FUNCTION_BLOCK FB_MotorControl
VAR_INPUT
	Run 			: BOOL; // Order to start running
	Ready			: BOOL; // Safety ok, system ok, doors ok
	Fast 			: BOOL;
	Faster			: BOOL;
	VFD_Running		: BOOL;
	VFD_Ready		: BOOL;
END_VAR
VAR_OUTPUT
	Q : BOOL;
	RUN_Order_VFD 	: BOOL;
	Fast_VFD		: BOOL;
	Faster_VFD		: BOOL;
	iRounds 	: INT;
	iRoundsMinute : INT;
	Gato 		: BOOL;
	Perro 		: BOOL;
	GatoCount 	: INT;
	PerroCount 	: INT;
	iStatus		: INT;
	iFault		: INT;
END_VAR
VAR
	
	Run_TRIG: R_TRIG;
	nMotorState: (NOT_READY, ALL_READY, RUNNING, STOP, ERROR);
	SwitchLeft_TRIG: R_TRIG;
	SwitchRight_TRIG: R_TRIG;
	Stopping_TON: TON;
END_VAR

// Rough outline:
// INPUT 24V: DIB 4 5 6 eli paikat 14 15 16
// 4 käy/seis, 5 vakionopeus 1, 6 vakionopeus 2
// Taajarilta viestiä että joko on käynnissä tai valmis, ei tiedä vielä

// OUTPUT: 20, 24 25 26
// 20 = DO1, VALMIS-signaali
// 24-26 = rele, 25 vaihtaa paikkaa

// Kaukosäätimellä napilla käynnistyy ja pysähtyy (valo syttyy tai sammuu)
// Kytkimellä nopeus 1 tai 2 (vilkuttaa myös nopeammin tai hitaammin)

// Yksi anturi olisi pyörässä kiinni laskemassa kierroksia
// Valoanturi seuraamassa kun kissa tai koira menee ohi

// Valmius ja moottori käy/ei käy keskustelu taajarin kanssa joko digitaalilähdön kautta (valmius ehkä?) ja relelähdön kautta (miten toimikaan? Pitiköhän syöttää virtaa keskelle)
//Inputit vois Triguina yhä käsitellä, vaikka Buttonboxistakin tulee triguja. Mikäli jostain muusta lähteestä tulee käskyjä niin onpahan triguja yhä

//==================
// 7.10.22
// Moottori pyörii, käskyjä liikkuu. nyt erikoiskäyttö -profiili taajarissa, mutta EEPROM vika unohtaa kaikki asetukset.
// IN 1,2 on käy/suunta nyt, ei jaksa vaihtaa paremmaksi. 3 on Fast, mutta IN 4 ei ole taajarissa kytketty (sitten olisi Faster)
// OUT (taajarista) ei nopeasti katsoen rekisteröidy PLC:ssä. Relelähtö varmaan vääri kytketty


A_ButtonHandling();

CASE nMotorState OF
	NOT_READY:	
		Q := FALSE;
		IF Ready THEN
		nMotorState := 1;
		END_IF

	ALL_READY:
		IF NOT Ready THEN
			nMotorState := 0;
		END_IF 

		IF Run_TRIG.Q THEN
			Q := TRUE;
			nMotorState := 2;		
		END_IF
		
	RUNNING:
		IF NOT Ready THEN
			nMotorState := 0;
		END_IF 
		
		IF Run_TRIG.Q THEN
			Q := FALSE;
			nMotorState := 3;
		END_IF
	STOP:
		Stopping_TON(IN:=TRUE , PT:=T#1S , Q=> , ET=> );
		IF Stopping_TON.Q THEN
			Stopping_TON(IN:=FALSE);
				nMotorState := 0;
		END_IF
	
	ERROR:
	
		
END_CASE

M_VariableChanges();

ACTION A_ButtonHandling:
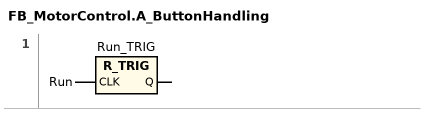
// NETWORK 1
Run_TRIG(CLK := Run); // R_TRIG
END_ACTION

METHOD M_VariableChanges : BOOL
VAR_INPUT
END_VAR

RUN_Order_VFD := Q;
Fast_VFD 	:= Fast;
Faster_VFD 	:= Faster;
iStatus 	:= nMotorState;
iFault 		:= 0;
END_METHOD

END_FUNCTION_BLOCK

(* stored: Version 1.1.0.1, ProductVersion 3.1.4024.10
   POU FB_MotorControl: Id {da1577ed-8fa5-451c-b384-ecb49194f3dd}, SpecialFunc None
   Action A_ButtonHandling: Id {42611ca4-32ab-4a2e-879d-1b2734acb427}
   Method M_VariableChanges: Id {25e58fda-e379-4634-b5e8-87a1ef140024} *)
